// TIA Portal V20 export
// export: Created 2025-12-01T14:56:21.0091572Z, ExportSetting None, DisplayName Totally Integrated Automation Portal, DisplayVersion V20 Update 3, DisplayName TIA Portal Openness, DisplayVersion V20 Update 3, DisplayName TIA Portal Version Control Interface, DisplayVersion V20 Update 3, DisplayName STEP 7 Professional, DisplayVersion V20 Update 3, DisplayName STEP 7 Safety, DisplayVersion V20 Update 2, DisplayName WinCC Basic/Comfort/Advanced, DisplayVersion V20 Update 3, DisplayName WinCC Professional, DisplayVersion V20 Update 3, DisplayName WinCC Unified, DisplayVersion V20 Update 3
TYPE "Temporizadores_flujos_mesa"
   STRUCT
      MAUX_INICIO_REGISTRO : Bool;
      MAUX_FIN_REGISTRO : Bool;
      NUM_REGISTRO_ACTUAL { ExternalAccessible := 'False'; ExternalVisible := 'False'; ExternalWritable := 'False'} : Int;
      TMP_Etapas_Carga_E0 { S7_SetPoint := 'True'} : TONR_TIME;
      TMP_Etapas_Carga_E1 { S7_SetPoint := 'True'} : TONR_TIME;
      TMP_Etapas_Carga_E2 { S7_SetPoint := 'True'} : TONR_TIME;
      TMP_Etapas_Carga_E3 { S7_SetPoint := 'True'} : TONR_TIME;
      TMP_Etapas_Carga_E4 { S7_SetPoint := 'True'} : TONR_TIME;
      TMP_Etapas_Descarga_S0 { S7_SetPoint := 'True'} : TONR_TIME;
      TMP_Etapas_Descarga_S1 { S7_SetPoint := 'True'} : TONR_TIME;
      TMP_Etapas_Descarga_S2 { S7_SetPoint := 'True'} : TONR_TIME;
      TMP_Etapas_Descarga_S3 { S7_SetPoint := 'True'} : TONR_TIME;
      TMP_Etapas_Descarga_S4 { S7_SetPoint := 'True'} : TONR_TIME;
      TMP_Etapa_Cargada { S7_SetPoint := 'True'} : TONR_TIME;
      TMP_AvanceRetroceso_Cadenas { S7_SetPoint := 'True'} : TONR_TIME;
      TMP_AvanceRetroceso_Rodillos { S7_SetPoint := 'True'} : TONR_TIME;
      TMP_Giro { S7_SetPoint := 'True'} : TONR_TIME;
      TMP_Subir_Transfer { S7_SetPoint := 'True'} : TONR_TIME;
      TMP_Bajar_Transfer { S7_SetPoint := 'True'} : TONR_TIME;
   END_STRUCT;
END_TYPE
